// TwinCAT 3 PLC project XtsTransport
// Title: XTS Transport
// Author: D.Hauer
// ProjectVersion: 0.0.1
// Description: basic functionblocks for building XTS transport
// ProgramVersion: 3.1.4024.0
// libraries:
//   Tc2_Math, * (Beckhoff Automation GmbH)
//   Tc2_MC2, * (Beckhoff Automation GmbH)
//   Tc2_Standard, * (Beckhoff Automation GmbH)
//   Tc2_System, * (Beckhoff Automation GmbH)
//   Tc2_Utilities, * (Beckhoff Automation GmbH)
//   Tc3_McCollisionAvoidance, * (Beckhoff Automation GmbH)
//   Tc3_McCoordinatedMotion, * (Beckhoff Automation GmbH)
//   Tc3_Module, * (Beckhoff Automation GmbH)
//   Tc3_XTS_Utility, * (Beckhoff Automation GmbH)
//   VisuDialogs, * (System)
// project tree:
//   / GlobalTextList.TcGTLO, GROUP.TcPOU (not stored), GROUP_VISU.TcVIS, MAIN.TcPOU (not stored), MOVER.TcPOU (not stored), MOVER_VISU.TcVIS (not stored), PlcTask.TcTTO (not stored), Visualization Manager.TcVMO (not stored)
//   XTS/CaGroup/ FB_CaGroup.TcPOU
//   XTS/CaGroup/types/ E_GROUP_CHECK.TcDUT (not stored), ST_GROUP_INFO.TcDUT (not stored)
//   XTS/ GVL_XTS.TcGVL, XTS_Parameter.TcGVL (not stored)
//   XTS/Mover/ fb_Mover.TcPOU (not stored)
//   XTS/Mover/types/ E_MOVER_CTRL.TcDUT (not stored), E_MOVER_STATE.TcDUT (not stored), ST_GEAR_DATA.TcDUT (not stored), ST_MOVER_INFO.TcDUT (not stored), ST_MOVE_DATA.TcDUT (not stored)
//   XTS/_types/ E_PROGRESS.TcDUT (not stored)

// ---- XTS/GVL_XTS.TcGVL
{attribute 'qualified_only'}
VAR_GLOBAL
  //---------------------------------------------------------------------------
  // Collision avoidance group CA
  //
  // - add mover to group
  // - build group
  // - clear group
  CaGroup         : FB_CaGroup;

  // caclic mapping to MOTION/Objects/CaGroup 
  CaGroupRef      : Tc3_McCoordinatedMotion.AXES_GROUP_REF;

  // Info data from CaGroup FB
  CaGroupInfo     : ST_GROUP_INFO;
  //---------------------------------------------------------------------------

  //---------------------------------------------------------------------------
  // MC2 encapsulation, CA movement
  Mover           : ARRAY[1..MAX_MOVER] OF fb_Mover;
  LastPosition    : ARRAY[1..MAX_MOVER] OF LREAL;
  LastGap         : ARRAY[1..MAX_MOVER] OF LREAL;

  MoverInfo       : ARRAY[1..MAX_MOVER] OF ST_MOVER_INFO;

  MoveData        : ARRAY[1..MAX_MOVER] OF ST_MOVE_DATA;
  GearData        : ARRAY[1..MAX_MOVER] OF ST_GEAR_DATA;
  
  // cyclic mapping to MOTION/Axes
  AxisRefMover    : ARRAY[1..MAX_MOVER] OF Tc2_MC2.AXIS_REF;
  //---------------------------------------------------------------------------
END_VAR

// ---- XTS/CaGroup/FB_CaGroup.TcPOU
//---------------------------------------------------------------------------------------------------------------
//
//  HAUD 2023.12.13
//
//
//  fb_CaGroup
//  - handles CA group states
//  - add mover to group
//  - remove mover from group
//  - clear group error
//  - startup procedure for getting group ready to work
//
//
//  VAR INPUT / OUTPUT --> see properties
//
//---------------------------------------------------------------------------------------------------------------//
// This SOFTWARE is provided as an Exemple by THE PROVIDER "as is" and "with all faults." THE PROVIDER makes no  //
// representations or warranties of any kind concerning the safety, suitability, lack of viruses, inaccuracies,  //
// typographical errors, or other harmful components of this SOFTWARE. There are inherent dangers in the use of  //
// any software, and you are solely responsible for determining whether this SOFTWARE is compatible with your    //
// equipment and other software installed on your equipment. You are also solely responsible for the protection  //
// of your equipment and backup of your data, and THE PROVIDER will not be liable for any damages you may suffer //
// in connection with using, modifying, or distributing this SOFTWARE.                                           //
//---------------------------------------------------------------------------------------------------------------//
FUNCTION_BLOCK FB_CaGroup	//IMPLEMENTS I_CaGroup
VAR
  _eCheck                     : E_GROUP_CHECK;
  _bError                     : BOOL;

  _GroupRef                   : REFERENCE TO Tc3_McCoordinatedMotion.AXES_GROUP_REF;
  _GroupCommon                : MCTOPLC_GROUP_COMMON_PART;

  _AxisRefMover               : REFERENCE TO ARRAY[1..MAX_MOVER] OF Tc2_MC2.AXIS_REF;


  // MC2 function block for halting all motion commands on mover before switching off group
  _fbHalt                     : ARRAY[1..MAX_MOVER] OF Tc2_MC2.MC_Halt;
  _fbReset                    : ARRAY[1..MAX_MOVER] OF Tc2_MC2.MC_Reset;

  // CA group fb instances
  _fbAddAxisGroup             : ARRAY[1..MAX_MOVER] OF Tc3_McCoordinatedMotion.MC_AddAxisToGroup;
  _fbRemoveAxisGroup          : ARRAY[1..MAX_MOVER] OF Tc3_McCoordinatedMotion.MC_RemoveAxisFromGroup;

  _fbGroupDisable             : Tc3_McCoordinatedMotion.MC_GroupDisable;
  _fbGroupEnable              : Tc3_McCoordinatedMotion.MC_GroupEnable;
  _fbGroupErrorRead           : Tc3_McCoordinatedMotion.MC_GroupReadError;
  _fbGroupStatusRead          : Tc3_McCoordinatedMotion.MC_GroupReadStatus;
  _fbGroupReset               : Tc3_McCoordinatedMotion.MC_GroupReset;

  _stGroupInfo                : ST_GROUP_INFO;  // additional bits about the state of the CA group

  _rtrigGroupStatusRead,
  _rtrigGroupErrorRead        : Tc2_Standard.R_TRIG;


END_VAR

METHOD AddAll : E_PROGRESS
VAR_INPUT
  Execute     : BOOL;
END_VAR
VAR_INST
  _nErrorId   : UDINT;
  _eState     : E_PROGRESS;

  _nMover     : UINT;
END_VAR
IF NOT Execute THEN _eState     := E_PROGRESS.PROGRESS_INIT; END_IF 
IF NOT Check() THEN AddAll := E_PROGRESS.PROGRESS_ERROR; RETURN; END_IF


CASE _eState
OF
  E_PROGRESS.PROGRESS_INIT:
    IF Execute
    THEN
      _nErrorId               := 0;
      _nMover                 := 1;
      _eState                 := E_PROGRESS.PROGRESS_BUSY;
    END_IF
END_CASE
//-----------------------------------------------------------------------------
//-----------------------------------------------------------------------------
CASE _eState
OF
  E_PROGRESS.PROGRESS_BUSY:
    _eState                   := E_PROGRESS.PROGRESS_PREPARE;
    _fbAddAxisGroup[_nMover](
                AxesGroup     := _GroupRef, 
                Axis          := _AxisRefMover[_nMover], 
                Execute       := FALSE, 
                IdentInGroup  := UDINT_TO_IDENTINGROUP(_AxisRefMover[_nMover].NcToPlc.AxisId));
END_CASE
//-----------------------------------------------------------------------------
//-----------------------------------------------------------------------------
CASE _eState
OF
  E_PROGRESS.PROGRESS_PREPARE:
    _fbAddAxisGroup[_nMover](
                AxesGroup     := _GroupRef, 
                Axis          := _AxisRefMover[_nMover], 
                Execute       := TRUE, 
                IdentInGroup  := UDINT_TO_IDENTINGROUP(_AxisRefMover[_nMover].NcToPlc.AxisId));

    IF (_fbAddAxisGroup[_nMover].Error)
    THEN
      _eState                 := E_PROGRESS.PROGRESS_ERROR;
      _nErrorId               := _fbAddAxisGroup[_nMover].ErrorId;

    ELSIF (_fbAddAxisGroup[_nMover].Done)
    THEN
      _eState                 := E_PROGRESS.PROGRESS_CHECK;
    END_IF
END_CASE
//-----------------------------------------------------------------------------
//-----------------------------------------------------------------------------
CASE _eState
OF
  E_PROGRESS.PROGRESS_CHECK:
    _eState                   := E_PROGRESS.PROGRESS_OCCUPIED;
    _fbAddAxisGroup[_nMover](
                AxesGroup     := _GroupRef, 
                Axis          := _AxisRefMover[_nMover], 
                Execute       := FALSE, 
                IdentInGroup  := UDINT_TO_IDENTINGROUP(_AxisRefMover[_nMover].NcToPlc.AxisId));
END_CASE
//-----------------------------------------------------------------------------
//-----------------------------------------------------------------------------
CASE _eState
OF
  E_PROGRESS.PROGRESS_OCCUPIED:
    _nMover                   := _nMover + 1;

    IF NOT (_nMover > MAX_MOVER)
    THEN
      _eState                 := E_PROGRESS.PROGRESS_BUSY;
    ELSE
      _eState                 := E_PROGRESS.PROGRESS_DONE;
    END_IF
END_CASE
//-----------------------------------------------------------------------------
//-----------------------------------------------------------------------------

AddAll                   := _eState;
END_METHOD

PROPERTY AxisRef : REFERENCE TO ARRAY[1..MAX_MOVER] OF Tc2_MC2.AXIS_REF
SET
_AxisRefMover REF= AxisRef;
END_SET
END_PROPERTY

METHOD PROTECTED Check : BOOL

IF NOT __ISVALIDREF(_GroupRef)
THEN
  _eCheck                     := E_GROUP_CHECK.CHECK_GROUP_REF_INVALID;
  RETURN;
END_IF

IF NOT __ISVALIDREF(_AxisRefMover)
THEN
  _eCheck                     := E_GROUP_CHECK.CHECK_AXIS_REF_INVALID;
  RETURN;
END_IF

_eCheck                       := E_GROUP_CHECK.CHECK_DONE;
Check                         := TRUE;
END_METHOD

METHOD Disable : E_PROGRESS
VAR_INPUT
  Execute     : BOOL;
END_VAR
VAR_INST
  _nErrorId   : UDINT;
  _eState     : E_PROGRESS;

  _nMover     : UINT;
END_VAR
IF NOT Execute THEN _eState       := E_PROGRESS.PROGRESS_INIT; END_IF 
IF NOT Check() THEN Disable  := E_PROGRESS.PROGRESS_ERROR; RETURN; END_IF


CASE _eState
OF
  E_PROGRESS.PROGRESS_INIT:
    IF Execute
    THEN
      _nErrorId               := 0;
      _nMover                 := 1;
      _eState                 := E_PROGRESS.PROGRESS_BUSY;
    END_IF
END_CASE
//-----------------------------------------------------------------------------
//-----------------------------------------------------------------------------
CASE _eState
OF
  E_PROGRESS.PROGRESS_BUSY:
    _eState                   := E_PROGRESS.PROGRESS_PREPARE;
    _fbGroupDisable(
              AxesGroup       := _GroupRef, 
              Execute         := FALSE); 
END_CASE
//-----------------------------------------------------------------------------
//-----------------------------------------------------------------------------
CASE _eState
OF
  E_PROGRESS.PROGRESS_PREPARE:
    _fbGroupDisable(
              AxesGroup       := _GroupRef, 
              Execute         := TRUE); 

    IF (_fbGroupDisable.Error)
    THEN
      _eState                 := E_PROGRESS.PROGRESS_ERROR;
      _nErrorId               := _fbGroupDisable.ErrorId;
      _fbGroupDisable(
              AxesGroup       := _GroupRef, 
              Execute         := FALSE); 


    ELSIF (_fbGroupDisable.Done)
    THEN
      _eState                 := E_PROGRESS.PROGRESS_DONE;
      _fbGroupDisable(
              AxesGroup       := _GroupRef, 
              Execute         := FALSE); 
    END_IF
END_CASE
//-----------------------------------------------------------------------------
//-----------------------------------------------------------------------------

Disable                  := _eState;
END_METHOD

METHOD Enable : E_PROGRESS
VAR_INPUT
  Execute     : BOOL;
END_VAR
VAR_INST
  _nErrorId   : UDINT;
  _eState     : E_PROGRESS;

  _nMover     : UINT;
END_VAR
IF NOT Execute THEN _eState       := E_PROGRESS.PROGRESS_INIT; END_IF 
IF NOT Check() THEN Enable   := E_PROGRESS.PROGRESS_ERROR; RETURN; END_IF


CASE _eState
OF
  E_PROGRESS.PROGRESS_INIT:
    IF Execute
    THEN
      _nErrorId               := 0;
      _nMover                 := 1;
      _eState                 := E_PROGRESS.PROGRESS_BUSY;
    END_IF
END_CASE
//-----------------------------------------------------------------------------
//-----------------------------------------------------------------------------
CASE _eState
OF
  E_PROGRESS.PROGRESS_BUSY:
    _eState                   := E_PROGRESS.PROGRESS_PREPARE;
    _fbGroupEnable(
                AxesGroup     := _GroupRef, 
                Execute       := FALSE);
END_CASE
//-----------------------------------------------------------------------------
//-----------------------------------------------------------------------------
CASE _eState
OF
  E_PROGRESS.PROGRESS_PREPARE:
    _fbGroupEnable(
                AxesGroup     := _GroupRef, 
                Execute       := TRUE);

    IF (_fbGroupEnable.Error)
    THEN
      _eState                 := E_PROGRESS.PROGRESS_ERROR;
      _nErrorId               := _fbGroupEnable.ErrorId;

      _fbGroupEnable(
                AxesGroup     := _GroupRef, 
                Execute       := FALSE);

    ELSIF (_fbGroupEnable.Done)
    THEN
      _eState                 := E_PROGRESS.PROGRESS_DONE;

      _fbGroupEnable(
                AxesGroup     := _GroupRef, 
                Execute       := FALSE);
    END_IF
END_CASE
//-----------------------------------------------------------------------------
//-----------------------------------------------------------------------------

Enable                   := _eState;
END_METHOD

PROPERTY GroupInfo : reference to ST_GROUP_INFO
GET
GroupInfo REF= _stGroupInfo;
END_GET
END_PROPERTY

PROPERTY GroupRef : reference to Tc3_McCoordinatedMotion.AXES_GROUP_REF
GET
GroupRef REF= _GroupRef;
END_GET
SET
_GroupRef REF= GroupRef;
END_SET
END_PROPERTY

METHOD InfoCycle : DWORD
VAR_INPUT
  Enable          : BOOL;
END_VAR
VAR_INST
  _nErrorIdADS,
  _nErrorIdRead   : UDINT;
END_VAR
IF NOT Check() THEN RETURN; END_IF


//-----------------------------------------------------------------------------------------------
// cyclic CA group
//-----------------------------------------------------------------------------------------------
_fbGroupStatusRead(
              AxesGroup                     := _GroupRef, 
              Enable                        := Enable, 
              Valid                         => _stGroupInfo.GroupStatusValid, 
              Busy                          => _stGroupInfo.GroupStatusBusy, 
              GroupMoving                   => _stGroupInfo.GroupMoving, 
              GroupHoming                   => _stGroupInfo.GroupHoming, 
              GroupErrorStop                => _stGroupInfo.GroupErrorStop, 
              GroupNotReady                 => _stGroupInfo.GroupNotReady, 
              GroupStandby                  => _stGroupInfo.GroupStandby, 
              GroupStopping                 => _stGroupInfo.GroupStopping, 
              GroupDisabled                 => _stGroupInfo.GroupDisabled, 
              AllAxesStanding               => _stGroupInfo.AllAxesStanding, 
              ConstantVelocity              => _stGroupInfo.ConstantVelocity, 
              Accelerating                  => _stGroupInfo.Accelerating, 
              Decelerating                  => _stGroupInfo.Decelerating, 
              InPosition                    => _stGroupInfo.InPosition, 
              Error                         => , 
              ErrorId                       => );

_fbGroupErrorRead(
              AxesGroup                     := _GroupRef, 
              Enable                        := Enable, 
              ErrorId                       => , 
              GroupErrorId                  => );


_stGroupInfo.AxisCount := _GroupRef.NcToPlc.CA.Common.GroupAxesCount;		  
			  
// fetch group error
_rtrigGroupStatusRead(CLK                   := (_stGroupInfo.GroupError OR
                                                _stGroupInfo.GroupErrorStop));
IF _rtrigGroupStatusRead.Q
THEN
  _stGroupInfo.GroupError   := _bError      := TRUE;
  _stGroupInfo.GroupErrorId                 := _fbGroupErrorRead.GroupErrorId;
END_IF

// fetch internal fb error
_rtrigGroupErrorRead(CLK                    := _fbGroupErrorRead.Error);
IF _rtrigGroupErrorRead.Q
THEN
  _nErrorIdADS                              := _fbGroupErrorRead.ErrorId;
END_IF
END_METHOD

METHOD McHaltAll : E_PROGRESS
VAR_INPUT
  Execute       : BOOL;
END_VAR
VAR_INST
  _nErrorId     : UDINT;
  _eState       : E_PROGRESS;

  _nMover       : UINT;
END_VAR
IF NOT Execute 
THEN 
	_eState     := E_PROGRESS.PROGRESS_INIT; 
END_IF 
IF NOT Check() 
THEN 
	McHaltAll   := E_PROGRESS.PROGRESS_ERROR; 
	RETURN; 
END_IF


CASE _eState
OF
  E_PROGRESS.PROGRESS_INIT:
    IF Execute
    THEN
      _nErrorId               := 0;
      _nMover                 := 1;
      _eState                 := E_PROGRESS.PROGRESS_BUSY;
    END_IF
END_CASE

//-----------------------------------------------------------------------------
//-----------------------------------------------------------------------------
CASE _eState
OF
  E_PROGRESS.PROGRESS_BUSY:
    _eState                   := E_PROGRESS.PROGRESS_PREPARE;
    FOR _nMover := 1 TO MAX_MOVER
    DO
      _fbHalt[_nMover](
                Axis          := _AxisRefMover[_nMover], 
                Execute       := FALSE, 
                Deceleration  := 15_000, 
                Jerk          := 150_000, 
                BufferMode    := MC_BufferMode.MC_Aborting,
                Error=> , 
                ErrorID=> );
    END_FOR
END_CASE

//-----------------------------------------------------------------------------
//-----------------------------------------------------------------------------
CASE _eState
OF
  E_PROGRESS.PROGRESS_PREPARE:
    _GroupCommon              := _GroupRef.NcToPlc.Common;
    IF (_GroupCommon.GroupStatus.Flags.AllAxesStanding)
    THEN
      _eState                 := E_PROGRESS.PROGRESS_CHECK;
    END_IF

    FOR _nMover := 1 TO MAX_MOVER
    DO
      _fbHalt[_nMover](
                Axis          := _AxisRefMover[_nMover], 
                Execute       := TRUE, 
                Deceleration  := 15_000, 
                Jerk          := 150_000, 
                BufferMode    := MC_BufferMode.MC_Aborting,
                Error=> , 
                ErrorID=>);
      IF (_fbHalt[_nMover].Error)
      THEN
        _nErrorId             := _fbHalt[_nMover].ErrorID;
        _eState               := E_PROGRESS.PROGRESS_ERROR;
        EXIT;
      END_IF
    END_FOR
END_CASE

//-----------------------------------------------------------------------------
//-----------------------------------------------------------------------------
CASE _eState
OF
  E_PROGRESS.PROGRESS_CHECK:
    _eState                   := E_PROGRESS.PROGRESS_DONE;
    FOR _nMover := 1 TO MAX_MOVER
    DO
      _fbHalt[_nMover](
                Axis          := _AxisRefMover[_nMover], 
                Execute       := FALSE, 
                Deceleration  := 15_000, 
                Jerk          := 150_000, 
                BufferMode    := MC_BufferMode.MC_Aborting,
                Error=> , 
                ErrorID=> );
    END_FOR
END_CASE

//-----------------------------------------------------------------------------
//-----------------------------------------------------------------------------

McHaltAll                     := _eState;
END_METHOD

METHOD McResetAll : E_PROGRESS
VAR_INPUT
  Execute       : BOOL;
END_VAR
VAR_INST
  _nErrorId     : UDINT;
  _eState       : E_PROGRESS;

  _nMover       : UINT;
END_VAR
IF NOT Execute THEN _eState     := E_PROGRESS.PROGRESS_INIT; END_IF 
IF NOT Check() THEN McResetAll  := E_PROGRESS.PROGRESS_ERROR; RETURN; END_IF


CASE _eState
OF
  E_PROGRESS.PROGRESS_INIT:
    IF Execute
    THEN
      _nErrorId               := 0;
      _nMover                 := 1;
      _eState                 := E_PROGRESS.PROGRESS_BUSY;
    END_IF
END_CASE
//-----------------------------------------------------------------------------
//-----------------------------------------------------------------------------
CASE _eState
OF
  E_PROGRESS.PROGRESS_BUSY:
    _eState                   := E_PROGRESS.PROGRESS_PREPARE;
    FOR _nMover := 1 TO MAX_MOVER
    DO
      _fbReset[_nMover](
                Axis          := _AxisRefMover[_nMover], 
                Execute       := FALSE);
    END_FOR
END_CASE
//-----------------------------------------------------------------------------
//-----------------------------------------------------------------------------
CASE _eState
OF
  E_PROGRESS.PROGRESS_PREPARE:
    _GroupCommon              := _GroupRef.NcToPlc.Common;
    IF (_GroupCommon.GroupStatus.Flags.AllAxesStanding)
    THEN
      _eState                 := E_PROGRESS.PROGRESS_CHECK;
    END_IF

    FOR _nMover := 1 TO MAX_MOVER
    DO
      _fbReset[_nMover](
                Axis          := _AxisRefMover[_nMover], 
                Execute       := TRUE);

      IF (_fbReset[_nMover].Error)
      THEN
        _nErrorId             := _fbReset[_nMover].ErrorID;
        _eState               := E_PROGRESS.PROGRESS_ERROR;
        EXIT;
      END_IF
    END_FOR
END_CASE
//-----------------------------------------------------------------------------
//-----------------------------------------------------------------------------
CASE _eState
OF
  E_PROGRESS.PROGRESS_CHECK:
    _eState                   := E_PROGRESS.PROGRESS_DONE;
    FOR _nMover := 1 TO MAX_MOVER
    DO
      _fbReset[_nMover](
                Axis          := _AxisRefMover[_nMover], 
                Execute       := FALSE);
    END_FOR
END_CASE
//-----------------------------------------------------------------------------
//-----------------------------------------------------------------------------

McResetAll                    := _eState;
END_METHOD

METHOD RemoveAll : E_PROGRESS
VAR_INPUT
  Execute     : BOOL;
END_VAR
VAR_INST
  _nErrorId   : UDINT;
  _eState     : E_PROGRESS;

  _nMover     : UINT;
END_VAR
IF NOT Execute THEN _eState         := E_PROGRESS.PROGRESS_INIT; END_IF 
IF NOT Check() THEN RemoveAll  := E_PROGRESS.PROGRESS_ERROR; RETURN; END_IF


CASE _eState
OF
  E_PROGRESS.PROGRESS_INIT:
    IF Execute
    THEN
      _nErrorId               := 0;
      _nMover                 := 1;
      _GroupCommon            := _GroupRef.NcToPlc.Common;

      IF (_GroupCommon.GroupAxesCount > 0)
      THEN
        _eState               := E_PROGRESS.PROGRESS_BUSY;
      ELSE
        _eState               := E_PROGRESS.PROGRESS_DONE;
      END_IF
    END_IF
END_CASE
//-----------------------------------------------------------------------------
//-----------------------------------------------------------------------------
CASE _eState
OF
  E_PROGRESS.PROGRESS_BUSY:
    _eState                   := E_PROGRESS.PROGRESS_PREPARE;
    _fbRemoveAxisGroup[_nMover](
              AxesGroup       := _GroupRef, 
              Execute         := FALSE,
              IdentInGroup    := UDINT_TO_IDENTINGROUP(_AxisRefMover[_nMover].NcToPlc.AxisId));
END_CASE
//-----------------------------------------------------------------------------
//-----------------------------------------------------------------------------
CASE _eState
OF
  E_PROGRESS.PROGRESS_PREPARE:
    _fbRemoveAxisGroup[_nMover](
              AxesGroup       := _GroupRef, 
              Execute         := TRUE,
              IdentInGroup    := UDINT_TO_IDENTINGROUP(_AxisRefMover[_nMover].NcToPlc.AxisId));

    IF (_fbRemoveAxisGroup[_nMover].Error)
    THEN
      _eState                 := E_PROGRESS.PROGRESS_ERROR;
      _nErrorId               := _fbRemoveAxisGroup[_nMover].ErrorId;

    ELSIF (_fbRemoveAxisGroup[_nMover].Done)
    THEN
      _eState                 := E_PROGRESS.PROGRESS_CHECK;
    END_IF
END_CASE
//-----------------------------------------------------------------------------
//-----------------------------------------------------------------------------
CASE _eState
OF
  E_PROGRESS.PROGRESS_CHECK:
    _eState                   := E_PROGRESS.PROGRESS_OCCUPIED;
    _fbRemoveAxisGroup[_nMover](
              AxesGroup       := _GroupRef, 
              Execute         := FALSE,
              IdentInGroup    := UDINT_TO_IDENTINGROUP(_AxisRefMover[_nMover].NcToPlc.AxisId));
END_CASE
//-----------------------------------------------------------------------------
//-----------------------------------------------------------------------------
CASE _eState
OF
  E_PROGRESS.PROGRESS_OCCUPIED:
    _nMover                   := _nMover + 1;

    IF NOT (_nMover > MAX_MOVER)
    THEN
      _eState                 := E_PROGRESS.PROGRESS_BUSY;
    ELSE
      _eState                 := E_PROGRESS.PROGRESS_DONE;
    END_IF
END_CASE
//-----------------------------------------------------------------------------
//-----------------------------------------------------------------------------

RemoveAll                := _eState;
END_METHOD

METHOD Reset : E_PROGRESS
VAR_INPUT
  Execute     : BOOL;
END_VAR
VAR_INST
  _nErrorId   : UDINT;
  _eState     : E_PROGRESS;

  _nMover     : UINT;
END_VAR
IF NOT Execute 
THEN 
	_eState := E_PROGRESS.PROGRESS_INIT; 
END_IF 
IF NOT Check() 
THEN 
	Reset := E_PROGRESS.PROGRESS_ERROR; 
	RETURN; 
END_IF


CASE _eState
OF
  E_PROGRESS.PROGRESS_INIT:
    IF Execute
    THEN
      _nErrorId                 := 0;
      _nMover                   := 1;
      _stGroupInfo.GroupErrorId := 0;
      _stGroupInfo.GroupError   := FALSE;

      _eState                   := E_PROGRESS.PROGRESS_BUSY;
    END_IF
END_CASE
//-----------------------------------------------------------------------------
//-----------------------------------------------------------------------------
CASE _eState
OF
  E_PROGRESS.PROGRESS_BUSY:
    _eState                     := E_PROGRESS.PROGRESS_PREPARE;
    _fbGroupReset(
              AxesGroup         := _GroupRef, 
              Execute           := FALSE);
END_CASE
//-----------------------------------------------------------------------------
//-----------------------------------------------------------------------------
CASE _eState
OF
  E_PROGRESS.PROGRESS_PREPARE:
    _fbGroupReset(
              AxesGroup         := _GroupRef, 
              Execute           := TRUE);

    IF (_fbGroupReset.Error)
    THEN
      _eState                   := E_PROGRESS.PROGRESS_ERROR;
      _nErrorId                 := _fbGroupReset.ErrorId;
      _fbGroupReset(
              AxesGroup         := _GroupRef, 
              Execute           := FALSE); 


    ELSIF (_fbGroupReset.Done)
    THEN
      _eState                   := E_PROGRESS.PROGRESS_DONE;
      _fbGroupReset(
              AxesGroup         := _GroupRef, 
              Execute           := FALSE); 
    END_IF
END_CASE
//-----------------------------------------------------------------------------
//-----------------------------------------------------------------------------

Reset                           := _eState;
END_METHOD

END_FUNCTION_BLOCK

// ---- GlobalTextList.TcGTLO
TEXTLIST GlobalTextList
  294 = '%.2f'
  191 = '%d'
  918 = '%r'
  562 = 'AllAxisStanding'
  162 = 'AxisCount: %d'
  914 = 'ConstantVelocity'
  359 = 'Decelerating'
  846 = 'eCtrlMover: %d'
  598 = 'eStateMover'
  432 = 'eStateMover: %d'
  958 = 'GROUP.bGroupBuild'
  79 = 'GROUP.bGroupClear'
  159 = 'GROUP.bGroupEnable'
  48 = 'GroupDisabled'
  915 = 'GroupError'
  590 = 'GroupErrorDtop'
  158 = 'GroupErrorId'
  495 = 'GroupErrorId: %d'
  975 = 'GroupErrorStop'
  940 = 'GroupHoming'
  300 = 'GroupMoving'
  807 = 'GroupNotReady'
  438 = 'GroupStandby'
  226 = 'GroupStatusBusy'
  602 = 'GroupStatusHoming'
  967 = 'GroupStatusMoving'
  204 = 'GroupStatusValid'
  973 = 'GroupStopping'
  75 = 'Info Act Pods Modulo'
  453 = 'Info Act Pos'
  211 = 'Info Act Pos Absolute'
  586 = 'Info Act Pos Modulo'
  21 = 'Info Mover Avoiding Collision'
  282 = 'Info Mover Coupled'
  398 = 'Info Mover Enabled'
  751 = 'Info Mover Error'
  907 = 'Info Mover Standstill'
  480 = 'Info nError ID'
  922 = 'Info Target Pos Absolute'
  16 = 'Info Target Pos Modulo'
  616 = 'InPosition'
  349 = 'Mover Avoiding Collision'
  585 = 'Mover Coupled'
  664 = 'Mover Enabled'
  243 = 'Mover Error'
  520 = 'Mover Standstill'
  732 = 'nError ID'
  756 = 'nMoverSelected: %d'
  984 = 'Set '
  91 = 'Set Acceleration'
  399 = 'Set Delta'
  382 = 'Set Distance'
  757 = 'Set Gap'
  934 = 'Set Jerk'
  201 = 'Set Override'
  936 = 'Set Position'
  62 = 'Set Velocity'
END_TEXTLIST

// ---- GROUP_VISU.TcVIS
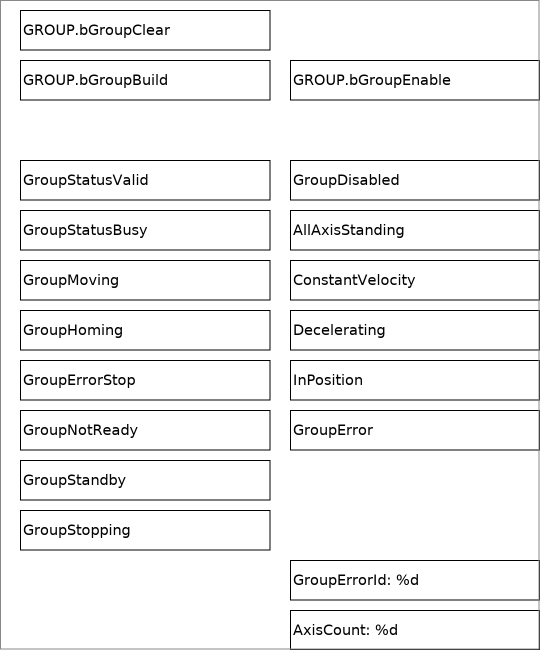
VISUALIZATION GROUP_VISU  // 540x650
    Rectangle (20,160 250x40), "GroupStatusValid", colour toggle: GVL_XTS.CaGroupInfo.GroupStatusValid
    Rectangle (20,210 250x40), "GroupStatusBusy", colour toggle: GVL_XTS.CaGroupInfo.GroupStatusBusy
    Rectangle (20,260 250x40), "GroupMoving", colour toggle: GVL_XTS.CaGroupInfo.GroupMoving
    Rectangle (20,310 250x40), "GroupHoming", colour toggle: GVL_XTS.CaGroupInfo.GroupHoming
    Rectangle (20,360 250x40), "GroupErrorStop", colour toggle: GVL_XTS.CaGroupInfo.GroupErrorStop
    Rectangle (20,410 250x40), "GroupNotReady", colour toggle: GVL_XTS.CaGroupInfo.GroupNotReady
    Rectangle (20,460 250x40), "GroupStandby", colour toggle: GVL_XTS.CaGroupInfo.GroupStandby
    Rectangle (20,510 250x40), "GroupStopping", colour toggle: GVL_XTS.CaGroupInfo.GroupStopping
    Rectangle (290,160 250x40), "GroupDisabled", colour toggle: GVL_XTS.CaGroupInfo.GroupDisabled
    Rectangle (290,210 250x40), "AllAxisStanding", colour toggle: GVL_XTS.CaGroupInfo.AllAxesStanding
    Rectangle (290,260 250x40), "ConstantVelocity", colour toggle: GVL_XTS.CaGroupInfo.ConstantVelocity
    Rectangle (290,310 250x40), "Decelerating", colour toggle: GVL_XTS.CaGroupInfo.Decelerating
    Rectangle (290,360 250x40), "InPosition", colour toggle: GVL_XTS.CaGroupInfo.InPosition
    Rectangle (290,410 250x40), "GroupError", colour toggle: GVL_XTS.CaGroupInfo.GroupError
    Rectangle (290,560 250x40), "GroupErrorId: %d", text variable: GVL_XTS.CaGroupInfo.GroupErrorId
    Rectangle (290,610 250x40), "AxisCount: %d", text variable: GVL_XTS.CaGroupInfo.AxisCount
    Rectangle (20,10 250x40), "GROUP.bGroupClear", colour toggle: GROUP.bGroupClear
    Rectangle (20,60 250x40), "GROUP.bGroupBuild", colour toggle: GROUP.bGroupBuild
    Rectangle (290,60 250x40), "GROUP.bGroupEnable", colour toggle: GROUP.bGroupEnable
END_VISUALIZATION
